FUNCTION_BLOCK UN_Machine100 EXTENDS FB_UN_Base IMPLEMENTS ITF_UN_Machine100
VAR_INPUT
END_VAR
VAR_OUTPUT
END_VAR
VAR
// Local var
	s_stMachineCommands				: ST_UN_Machine100_Cmd;	

// Config Struct
	s_stConfig						: ST_UN_Machine100_Config;

END_VAR

SUPER^();

METHOD PROTECTED _m_Alarms
SUPER^._m_Alarms();
END_METHOD

METHOD PROTECTED _m_Logic
SUPER^._m_Logic();
END_METHOD

METHOD PROTECTED _m_Modules
SUPER^._m_Modules();

// Example module
IF GVL_Area100.g_emLogicExample.p_itfAlarmCollector <> 0
	AND_THEN __ISVALIDREF(GVL_Area100.g_emLogicExample.p_itfAlarmCollector.p_rstConfig)
THEN
	GVL_Area100.g_emLogicExample.p_itfAlarmCollector.p_rstConfig.eSubstituteActionForPackML_Abort := E_Alarm_Actions.Stop;
END_IF
GVL_Area100.g_emLogicExample(
	i_bReqEnable		:= TRUE, 
	i_bReqReset			:= s_fbAlarmCollector.q_bReqReset,
	i_bStaSafetyOk		:= TRUE,
	i_bReqSimulationOn	:= s_fbSimulation.q_bStaOn,
	i_itfPackML_Parent	:= THIS^,
	i_itfAlarmCollector_Parent := s_fbAlarmCollector,
	i_stMachineCommands	:= s_stMachineCommands,
	i_itfPackML_StatusManager	:= i_itfPackML_StatusManager);



// Example module
GVL_Area100.g_emLogicExample2(
	i_bReqEnable		:= TRUE, 
	i_bReqReset			:= s_fbAlarmCollector.q_bReqReset,
	i_bStaSafetyOk		:= TRUE,
	i_bReqSimulationOn	:= s_fbSimulation.q_bStaOn,
	i_itfPackML_Parent	:= THIS^,
	i_itfAlarmCollector_Parent := s_fbAlarmCollector,
	i_stMachineCommands	:= s_stMachineCommands,
	i_itfPackML_StatusManager	:= i_itfPackML_StatusManager);

// Safety module
GVL_Area100.g_emSafety(
	i_bReqEnable		:= TRUE, 
	i_bReqReset			:= s_fbAlarmCollector.q_bReqReset,
	i_bStaSafetyOk		:= TRUE,
	i_bReqSimulationOn	:= s_fbSimulation.q_bStaOn,
	i_itfPackML_Parent	:= THIS^,
	i_itfAlarmCollector_Parent := s_fbAlarmCollector,
	i_stMachineCommands	:= s_stMachineCommands,
	i_itfPackML_StatusManager	:= i_itfPackML_StatusManager,
	q_bStaSafetyOk		=> );
END_METHOD

METHOD PUBLIC m_Main
SUPER^.m_Main();
END_METHOD

{attribute 'monitoring' := 'call'}
PROPERTY p_itfEmLogicExample : ITF_Hmi_ModuleBase
GET
p_itfEmLogicExample := GVL_Area100.g_emLogicExample;
END_GET
END_PROPERTY

{attribute 'monitoring' := 'call'}
PROPERTY p_itfEmSafety : ITF_Hmi_ModuleBase
GET
p_itfEmSafety := GVL_Area100.g_emSafety;
END_GET
END_PROPERTY

{attribute 'monitoring' := 'call'}
PROPERTY p_stConfig : REFERENCE TO ST_UN_Machine100_Config
GET
p_stConfig := s_stConfig;
END_GET
END_PROPERTY

END_FUNCTION_BLOCK

(* stored: Version 1.1.0.1, ProductVersion 3.1.4024.10
   POU UN_Machine100: Id {21e30d72-cc39-422e-8114-15c7abc2b847}, SpecialFunc None
   Folder Basic: Id {e89104c0-d33f-460a-aaf2-8953cfda25ab}
   Folder ITF_UN_Machine100: Id {993bc94f-48fd-4eea-942a-5c02e6ec715c}
   Method _m_Alarms: Id {8fa8464a-636c-46ee-9f13-6e7927953bcd}
   Method _m_Logic: Id {b95711e4-a3f3-4e91-9f55-7c0e3689d897}
   Method _m_Modules: Id {c15e282d-b76d-440b-8236-902bb4c31743}
   Method m_Main: Id {5738c138-41a1-473c-badd-a5f9691bbc49}
   Property p_itfEmLogicExample: Id {26224556-8538-4d9f-bcfc-37014048d854}
   Get Get: Id {623eaf14-77b2-40e4-839e-b7f0149cc8bb}
   Property p_itfEmSafety: Id {14512e0e-efa9-4836-b847-117ef07af89d}
   Get Get: Id {71671166-907c-4eeb-aa1b-fc56ebaa0f3e}
   Property p_stConfig: Id {10d73f7a-3734-442c-bff3-b37a394b7208}
   Get Get: Id {d0ae69ad-c446-4df5-88dc-fd69c355fa21} *)
